FUNCTION_BLOCK FillWindowFS_AR (* Colors a fill attributes object green/red (or any two colors) depending on whether an incoming AR value lies within a window *)
  (* Standard: ISO 11783-6; Description: Copyright (c) 2026 Meisterschulen am Ostbahnhof This program and the accompanying materials are made available under the terms of the Eclipse Public License 2.0 which is available at https://www.eclipse.org/legal/epl-2.0/ SPDX-License-Identifier: EPL-2.0 Wraps a single Q_FillAttributes instance (ISO 11783-6 F.32) that commands a FillAttributes object's colour. The incoming AR value is checked against [rWindowMin, rWindowMax] via F_WindowColor; u8ColorIn is sent while the value is inside the window, u8ColorOut otherwise. FillType and FillPatternId are fixed to solid colour (no pattern) - this block only ever changes the colour, not the fill style itself. *)
  (* Version 1.0, 2026-09-06, Franz Höpfinger, Meisterschulen am Ostbahnhof, initial API and implementation and/or initial documentation *)
  PACKAGE isobus::UT::Q;
  IMPORT isobus::UT::Q::Q_FillAttributes;
  IMPORT isobus::UT::Q::helpers::F_WindowColor;
  IMPORT isobus::UT::Q::const::IDs::ID_NULL;
  IMPORT isobus::UT::Q::const::colours::COLOR_GREEN;
  IMPORT isobus::UT::Q::const::colours::COLOR_RED;
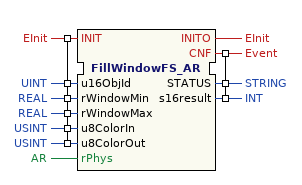
  EVENT_INPUT
    INIT : EInit WITH u16ObjId, rWindowMin, rWindowMax, u8ColorIn, u8ColorOut; (* Service Initialization *)
  END_EVENT
  EVENT_OUTPUT
    INITO : EInit; (* Initialization Confirm *)
    CNF WITH STATUS, s16result; (* Confirmation of Requested Service *)
  END_EVENT
  VAR_INPUT
    u16ObjId : UINT := ID_NULL; (* FillAttributes object ID to command *)
    rWindowMin : REAL; (* Lower bound of the window that shows u8ColorIn *)
    rWindowMax : REAL; (* Upper bound of the window that shows u8ColorIn *)
    u8ColorIn : USINT := COLOR_GREEN; (* Colour shown while the AR value is within [rWindowMin, rWindowMax] *)
    u8ColorOut : USINT := COLOR_RED; (* Colour shown while the AR value is outside [rWindowMin, rWindowMax] *)
  END_VAR
  VAR_OUTPUT
    STATUS : STRING; (* Service Status - passthrough from the internal Q_FillAttributes *)
    s16result : INT; (* retval - passthrough from the internal Q_FillAttributes *)
  END_VAR
  SOCKETS
    rPhys : adapter::types::unidirectional::AR; (* Value whose position relative to the window decides the colour *)
  END_SOCKETS
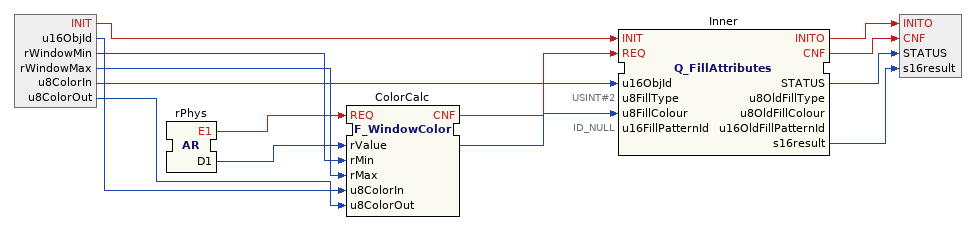
  FBS
    Inner : isobus::UT::Q::Q_FillAttributes(u8FillType := USINT#2, u16FillPatternId := ID_NULL);
    ColorCalc : isobus::UT::Q::helpers::F_WindowColor;
  END_FBS
  EVENT_CONNECTIONS
    INIT TO Inner.INIT;
    rPhys.E1 TO ColorCalc.REQ;
    ColorCalc.CNF TO Inner.REQ;
    Inner.INITO TO INITO;
    Inner.CNF TO CNF;
  END_CONNECTIONS
  DATA_CONNECTIONS
    u16ObjId TO Inner.u16ObjId;
    rPhys.D1 TO ColorCalc.rValue;
    rWindowMin TO ColorCalc.rMin;
    rWindowMax TO ColorCalc.rMax;
    u8ColorIn TO ColorCalc.u8ColorIn;
    u8ColorOut TO ColorCalc.u8ColorOut;
    ColorCalc. TO Inner.u8FillColour;
    Inner.STATUS TO STATUS;
    Inner.s16result TO s16result;
  END_CONNECTIONS
END_FUNCTION_BLOCK
